// Mitsubishi GX Works2 project: LD_tubewindingmachine   PLC: FX1N/FX1NC

PROGRAM MAIN
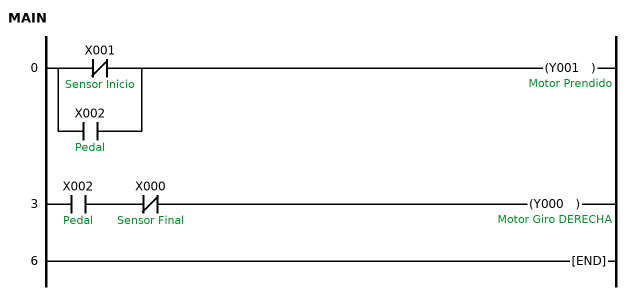
0     LDI     X001  ; Sensor Inicio
      OR      X002  ; Pedal
      OUT     Y001  ; Motor Prendido
3     LD      X002  ; Pedal
      ANI     X000  ; Sensor Final
      OUT     Y000  ; Motor Giro DERECHA
6     END
END_PROGRAM

// device comments not shown above
M0  ; M Giro Derecha
M1  ; M Final
M2  ; M Pedal
